Fanuc KAREL source: CNV_STR_TIME.kl

PROGRAM T
%NOLOCKGROUP
VAR
 v0 : STRING[40]
 v1 : INTEGER
BEGIN
 CNV_STR_TIME(v0, v1)
END T
